(* CoDeSys 2.3 export: DOWE.EXP *)

(* Data type in D7Timer *)
TYPE DoWE :
(
    Mon:=0,
    Tue,
    Wed,
    Thu,
    Fri,
    Sat,
    Sun
);
END_TYPE
